// TIA Portal V18 export
FUNCTION "RTDbasic" : Void   // FC10006, FBD
{ S7_Optimized_Access := 'TRUE' }
VERSION : 0.1
// stored: AutoNumber false, IsIECCheckEnabled false, SetENOAutomatically false, UDAEnableTagReadback false
   VAR_INPUT
      iInput : Int;
      rFilterValue : Real;
      rCalibration : Real;
      rDiv : Real;
   END_VAR
   VAR_OUTPUT
      rOutput : Real;
   END_VAR
BEGIN
END_FUNCTION
